TYPE Cilindro :
STRUCT
	posicion : REAL;
	extendido: BOOL;
	retraido: BOOL;
	parado: BOOL;
	extendiendo : BOOL;
	retrayendo: BOOL;
	regimen : REAL; //tnato por uno de apertura de válvula
END_STRUCT
END_TYPE

(* stored: Version 1.1.0.1, ProductVersion 3.1.4024.4
   DUT Cilindro: Id {35a15ef1-eecc-4376-af58-8f7421ae106e} *)
